// Provide logging 
FUNCTION_BLOCK FB_TcLogging IMPLEMENTS I_Logging
VAR_INPUT
	eLogLevel:				E_LogLevel:= E_LogLevel.Verbose;
END_VAR
VAR_OUTPUT
END_VAR
VAR
	iLogging:				I_Logging;
END_VAR

METHOD PUBLIC M_Attach : BOOL
VAR_INPUT
	iLogging:				I_Logging;
END_VAR
IF THIS^.iLogging = 0 THEN
	THIS^.iLogging:= iLogging;
	M_Attach:= TRUE;
ELSIF THIS^.iLogging = iLogging THEN
	// already inside
	M_Attach:= TRUE;
	RETURN;
ELSE
	// redirect to next logging function block
	THIS^.iLogging.M_Attach(iLogging);
END_IF
END_METHOD

METHOD PUBLIC M_Log : BOOL
VAR_INPUT
	stMessage:			ST_Message;
END_VAR
VAR
	fbMsg:				FB_TcMessage; 
	fbSourceInfo:		FB_TcSourceInfo;
END_VAR
IF THIS^.eLogLevel > eLogLevel THEN
	M_Log:= TRUE;
	RETURN;
END_IF

IF stMessage.bActive THEN

	fbSourceInfo.Clear();
	fbSourceInfo.sName:= stMessage.sSource;
	
	CASE stMessage.eLogLevel OF
		E_LogLevel.Verbose:
			fbMsg.CreateEx(TC_EVENTS.TcLogging.Verbose, fbSourceInfo); 	
	
		E_LogLevel.Info:
			fbMsg.CreateEx(TC_EVENTS.TcLogging.Info, fbSourceInfo); 
			
		E_LogLevel.Warning:		
			fbMsg.CreateEx(TC_EVENTS.TcLogging.Warning, fbSourceInfo); 
			
		E_LogLevel.Error:
			fbMsg.CreateEx(TC_EVENTS.TcLogging.Error, fbSourceInfo); 
			
		E_LogLevel.Critical:
			fbMsg.CreateEx(TC_EVENTS.TcLogging.Critical, fbSourceInfo); 
			
	END_CASE
	
	fbMsg.ipArguments.Clear().AddString(stMessage.sDefault);
	
	fbMsg.Send(stMessage.nTimestamp);

END_IF
END_METHOD

PROPERTY PUBLIC P_LogLevel : E_LogLevel
GET
P_LogLevel:= eLogLevel;
END_GET
SET
eLogLevel:= P_LogLevel;
END_SET
END_PROPERTY

END_FUNCTION_BLOCK

(* stored: Version 1.1.0.1
   POU FB_TcLogging: Id {a25dbc17-9138-425a-a854-e40fc76dd77c}, SpecialFunc None
   Method M_Attach: Id {1c8989a0-b07f-40c8-a8af-0456191e3a9c}
   Method M_Log: Id {577977a1-ae7e-4ffb-868f-fd739cd70e23}
   Property P_LogLevel: Id {afb8b02e-d604-4cf3-9992-3c35b57f3bbc}
   Get Get: Id {36c09c6b-534a-4aee-9f98-f1f60e550705}
   Set Set: Id {aee25470-c4df-4fee-aa5c-2c45b38c0a84} *)
